TYPE T_NEST_OFFSET : ARRAY[1..MAX_MOVER]        OF
                     ARRAY[1..MAX_STATION_NEST] OF LREAL;
END_TYPE

(* stored: Version 1.1.0.1
   DUT T_NEST_OFFSET: Id {22d19f2f-016e-4c25-ab96-d310fd9ee889} *)
